// TwinCAT 3 PLC project AbstactDataTypes
// ProgramVersion: 3.1.4022.7
// libraries:
//   Tc2_Standard, * (Beckhoff Automation GmbH)
//   Tc2_System, * (Beckhoff Automation GmbH)
//   Tc3_Module, * (Beckhoff Automation GmbH)
// project tree:
//   / PlcTask.TcTTO
//   POUs/Linked List/DUTs/ _ST_NODE_.TcDUT
//   POUs/Linked List/ HgFB_Linked_List.TcPOU
//   POUs/ MAIN.TcPOU
// real-time tasks:
//   TASK PlcTask: cycle T#10ms, priority 20, ADS port 350

CONFIGURATION AbstactDataTypes
    RESOURCE PLC ON TwinCAT3
        TASK PlcTask(INTERVAL := T#10ms, PRIORITY := 20);
        PROGRAM MAIN WITH PlcTask : MAIN;
    END_RESOURCE
END_CONFIGURATION

// ---- POUs/Linked List/DUTs/_ST_NODE_.TcDUT
{attribute 'enable_dynamic_creation'}
TYPE _ST_NODE_ :
STRUCT
	iData : INT;
	pNext : POINTER TO _ST_NODE_;
END_STRUCT
END_TYPE

// ---- POUs/MAIN.TcPOU
PROGRAM MAIN
VAR
	nState : BYTE;
	fbLinked_List : HgFB_Linked_List;
	aArray : ARRAY[0..10] OF INT;
END_VAR

 CASE nState OF 
	0: // Run fuctions once
		fbLinked_List.Init();
		fbLinked_List.Create(1);
		fbLinked_List.Create(2);
		fbLinked_List.Create(3);
		fbLinked_List.Display(aArray);
		
		
		nState := nState + 1;
END_CASE

END_PROGRAM

// ---- POUs/Linked List/HgFB_Linked_List.TcPOU
FUNCTION_BLOCK HgFB_Linked_List
VAR_INPUT
END_VAR
VAR_OUTPUT
END_VAR
VAR
	pHead :  POINTER TO _ST_NODE_;
	pTail :  POINTER TO _ST_NODE_;
END_VAR

// Adds an node to the end of the linked list
METHOD Create
VAR_INPUT
	iValue : INT;
END_VAR
VAR
	pTemp :  POINTER TO _ST_NODE_;
END_VAR
pTemp := __NEW(_ST_NODE_); 	// Allocate space in memory for a node.
pTemp^.iData := iValue;		// Assign Data to the new node.
pTemp^.pNext := NULL;		// Pointer to next node is NULL.
IF pHead = 0 THEN pHead := pTemp; pTail := pTemp; // If the pointer to the pHead is NULL then give it an address. The pTail address of the first node is the pHead.
ELSE  pTail^.pNext := pTemp; pTail := pTail^.pNext; END_IF // Point previous node's pNext to the address of pTemp and set pTail to pTemp.
END_METHOD

// Traverse the list to display each node
METHOD Display : BOOL
VAR_IN_OUT
	aList : ARRAY[*] OF INT;
END_VAR
VAR
	pCurrent :  POINTER TO _ST_NODE_;
	i : DINT;
END_VAR
//pCurrent := __NEW(_ST_NODE_); 	// Allocate space in memory for a node.
pCurrent := pHead;
i := LOWER_BOUND(aList, 1);
WHILE pCurrent <> 0 AND i < UPPER_BOUND(aList, 1) DO
	aList[i] := pCurrent^.iData;
	pCurrent := pCurrent^.pNext;
	i := i+1;
END_WHILE
END_METHOD

// Initializes or create an empty list
METHOD Init
pHead := NULL;
pTail := NULL;
END_METHOD

END_FUNCTION_BLOCK
